// TIA Portal V19 export
DATA_BLOCK "RO_1 DB"   // DB72
{ S7_Optimized_Access := 'FALSE' }
   VAR RETAIN
      OUTPUT : Struct
         "ABV-301" : Bool;
         "ABV-302" : Bool;
         "AGLV-301" : Bool;
         "AGLV-302" : Bool;
         "DP-703" : Bool;
         "DP-704" : Bool;
         "DP-705" : Bool;
         "RO-1 FEED PUMP" : Bool;
         "RO-1 HPP-301A" : Bool;
         "RO-1 HPP-301B" : Bool;
         "AGLV-301 RECIRC" : Bool;
         "AGLV-302 RECIRC" : Bool;
      END_STRUCT;
   END_VAR
BEGIN
END_DATA_BLOCK
